PROGRAM MAIN
VAR
	//strategy controller
	Strategy : BaseStrategyController; 

	//thermal networks
	CN : CoolingNetwork;
	HNLT_CN : HNLT_CN_Linkage;
	
	//cycle counter
	MAIN_CycleCount : UDINT;
    info  : GETCURTASKINDEX;
	test_output : REAL;
END_VAR

//Updated implementation
//Strategy(fTemperature_CN := Speicher.Pufferspeicher_Kaltwasser_195.Zustand.Temp_mitte);

Strategy(fTemperature_CN := CN.fTemperatureBufferStorage);

CN(fSetPointTemperature := Strategy.fTargetTemperature_CN,
	bSetStatusOn_eChiller := Strategy.bSetStatusOn_eChiller);

HNLT_CN(bSetStatusOn_HeatPump := Strategy.bSetStatusOn_HeatPump);
	
	
//test output for checking variable exchange between tasks with different cycle time
test_output := HeatCounter.test_output;
info();
MAIN_CycleCount := _TaskInfo[info.index].CycleCount;

END_PROGRAM

(* stored: Version 1.1.0.1, ProductVersion 3.1.4024.10
   POU MAIN: Id {9f33f5a0-2a24-4206-9468-c589128c5602}, SpecialFunc None *)
